{attribute 'GeneratedUsingTerminal: EL2521-0124-0018'}
{attribute addProperty BoxType "EL2521-0124-0018"}
{attribute addProperty Id "ControlAT %Q*Control_7786EF9F2Switch_on_valueAT %Q*UINT2Switch_off_valueAT %Q*UINT2"}
{attribute addProperty CRC "3446555870"}
{attribute addProperty Size "6"}
TYPE PLS_Control_compact_CD6E44DE EXTENDS OutputBase_10CEE7DE :
STRUCT
	{attribute addProperty Name "Control"}
	Control AT %Q* : Control_7786EF9F;
	{attribute addProperty Name "Switch_on_value"}
	Switch_on_value AT %Q* : UINT;
	{attribute addProperty Name "Switch_off_value"}
	Switch_off_value AT %Q* : UINT;
END_STRUCT
END_TYPE

(* stored: Version 1.2.0.0, ProductVersion 3.1.4024.11
   DUT PLS_Control_compact_CD6E44DE: Id {3b120002-c3e8-4d94-b90f-06cc659cae58} *)
